// TIA Portal V17 export
// export: Created 2024-08-09T12:50:01.0453715Z, ExportSetting WithDefaults, DisplayName Totally Integrated Automation Portal, DisplayVersion V17 Update 7, DisplayName TIA Portal Openness, DisplayVersion V17 Update 7, DisplayName TIA Portal Version Control Interface, DisplayVersion V17, DisplayName STEP 7 Professional, DisplayVersion V17 Update 7, DisplayName STEP 7 Safety, DisplayVersion V17 Update 6, DisplayName WinCC Professional, DisplayVersion V17 Update 7
DATA_BLOCK "DB_Aff_Def_Sup"   // DB5
VERSION : 0.1
// stored: AutoNumber true, DBAccessibleFromOPCUA true, DBAccessibleFromWebserver true, InstanceOfName Aff_Def_Sup, InstanceOfType FB
"Aff_Def_Sup"
   // VAR
   //    Aff_Def_Sup : Array[0..9] of "S_Defaut";
   //    Offset { ExternalAccessible := 'False'; ExternalVisible := 'False'; ExternalWritable := 'False'} : USInt;
   //    Num_Page : Int;
   //    Nbr_Msg : Int;
   // END_VAR
BEGIN
END_DATA_BLOCK
